// SIMATIC S7-200 project (STEP 7-Micro/WIN), CPU 226 REL 02.01

SYMBOL_TABLE 用户定义1
DDL              I0.0     // 压力继电器1
DDR              I0.1     // 压力继电器2
HP1              I0.2     // 正转水平位置
HP2              I0.3     // 反转水平位置
VP               I0.4     // 竖直位置
LMT1             I0.5     // 极限位置1
LMT2             I0.6     // 极限位置2
ERR              I0.7     // 急停或故障
TR               I1.2     // 正转点动
RT               I1.3     // 反转点动
HR1              I1.4     // 正转到水平
HR2              I1.5     // 反转到水平
TMP              M0.0     // 临时变量
FlagTR           M0.1     // 正转点动指令
FlagRT           M0.2     // 反转点动指令
FlagTRC          M0.3     // 正转到水平位置指令
FlagRTC          M0.4     // 反转到水平位置指令
EV1              Q0.0     // EV1
EV2              Q0.1     // EV2
EV3              Q0.2     // EV3
EV4              Q0.3     // EV4
EV5              Q0.4     // EV5
EV6              Q0.5     // EV6
EV7              Q0.6     // EV7
EV8              Q0.7     // EV8
AL1              Q1.0     // 翻转运行指示
AL2              Q1.1     // 系统运行指示
END_SYMBOL_TABLE

SYMBOL_TABLE S7-200 符号
Always_On        SM0.0    // 始终接通为 ON
First_Scan_On    SM0.1    // 仅第一个扫描周期中接通为 ON
END_SYMBOL_TABLE

ORGANIZATION_BLOCK 主程序:OB1
TITLE=程序注释
VAR
Flag_HR1_Enabled:BOOL;	// L0.0 一键转到水平位置1触发
Flag_HR2_Enabled:BOOL;	// L0.1 一键转到水平位置2触发
State_CurPosition:BYTE;	// LB1 当前位置
Cmd_TRC:BOOL;	// L2.0 
Cmd_RTC:BOOL;	// L2.1 
END_VAR
BEGIN
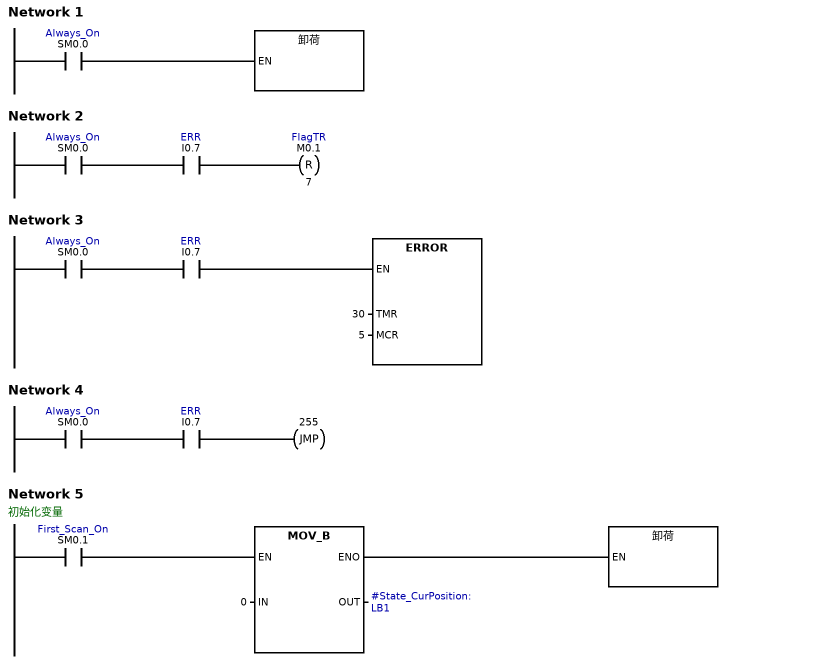
Network 1
LD     Always_On:SM0.0
CALL   卸荷:SBR0
Network 2
LD     Always_On:SM0.0
A      ERR:I0.7
R      FlagTR:M0.1, 7
Network 3
LD     Always_On:SM0.0
A      ERR:I0.7
CALL   ERROR:SBR8, 30, 5
Network 4
LD     Always_On:SM0.0
A      ERR:I0.7
JMP    255
Network 5
// 初始化变量
LD     First_Scan_On:SM0.1
MOVB   0, #State_CurPosition:LB1
AENO
CALL   卸荷:SBR0
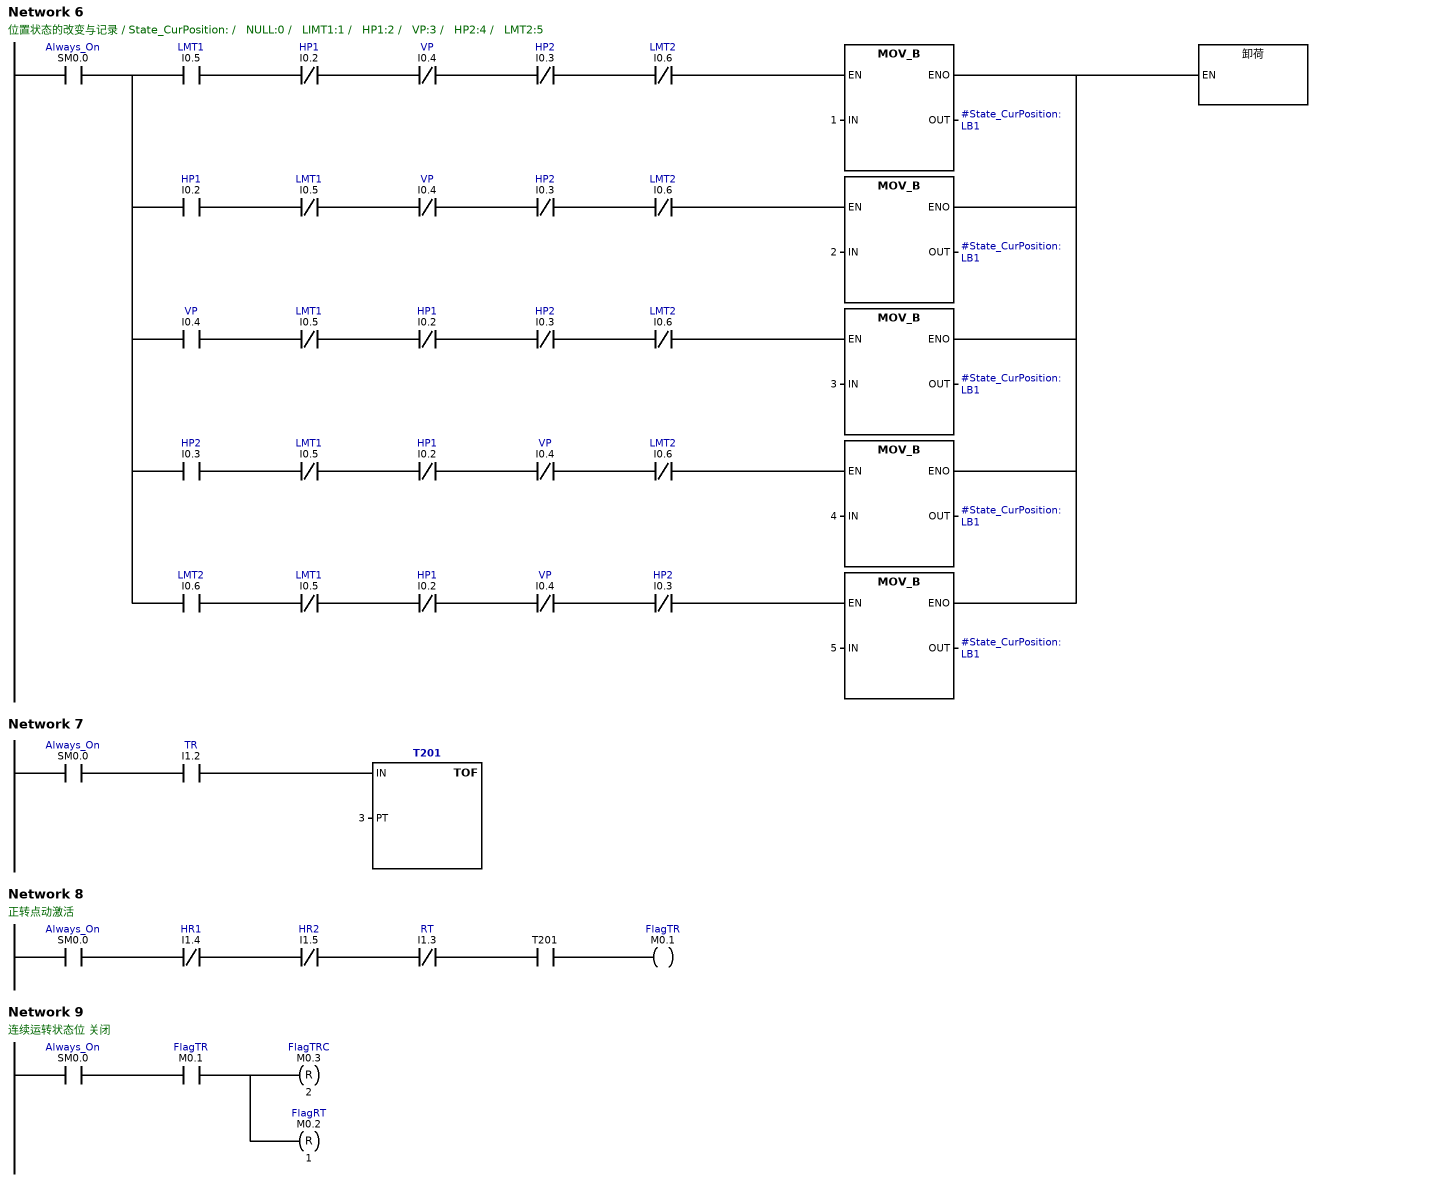
Network 6
// 位置状态的改变与记录
// State_CurPosition:
// 	NULL:0
// 	LIMT1:1
// 	HP1:2
// 	VP:3
// 	HP2:4
// 	LMT2:5
LD     Always_On:SM0.0
LPS
A      LMT1:I0.5
AN     HP1:I0.2
AN     VP:I0.4
AN     HP2:I0.3
AN     LMT2:I0.6
MOVB   1, #State_CurPosition:LB1
AENO
=      L63.7
LRD
A      HP1:I0.2
AN     LMT1:I0.5
AN     VP:I0.4
AN     HP2:I0.3
AN     LMT2:I0.6
MOVB   2, #State_CurPosition:LB1
AENO
O      L63.7
=      L63.6
LRD
A      VP:I0.4
AN     LMT1:I0.5
AN     HP1:I0.2
AN     HP2:I0.3
AN     LMT2:I0.6
MOVB   3, #State_CurPosition:LB1
AENO
O      L63.6
=      L63.5
LRD
A      HP2:I0.3
AN     LMT1:I0.5
AN     HP1:I0.2
AN     VP:I0.4
AN     LMT2:I0.6
MOVB   4, #State_CurPosition:LB1
AENO
O      L63.5
=      L63.4
LPP
A      LMT2:I0.6
AN     LMT1:I0.5
AN     HP1:I0.2
AN     VP:I0.4
AN     HP2:I0.3
MOVB   5, #State_CurPosition:LB1
AENO
O      L63.4
CALL   卸荷:SBR0
Network 7
LD     Always_On:SM0.0
A      TR:I1.2
TOF    T201, 3
Network 8
// 正转点动激活
LD     Always_On:SM0.0
AN     HR1:I1.4
AN     HR2:I1.5
AN     RT:I1.3
A      T201
=      FlagTR:M0.1
Network 9
// 连续运转状态位 关闭
LD     Always_On:SM0.0
A      FlagTR:M0.1
R      FlagTRC:M0.3, 2
R      FlagRT:M0.2, 1
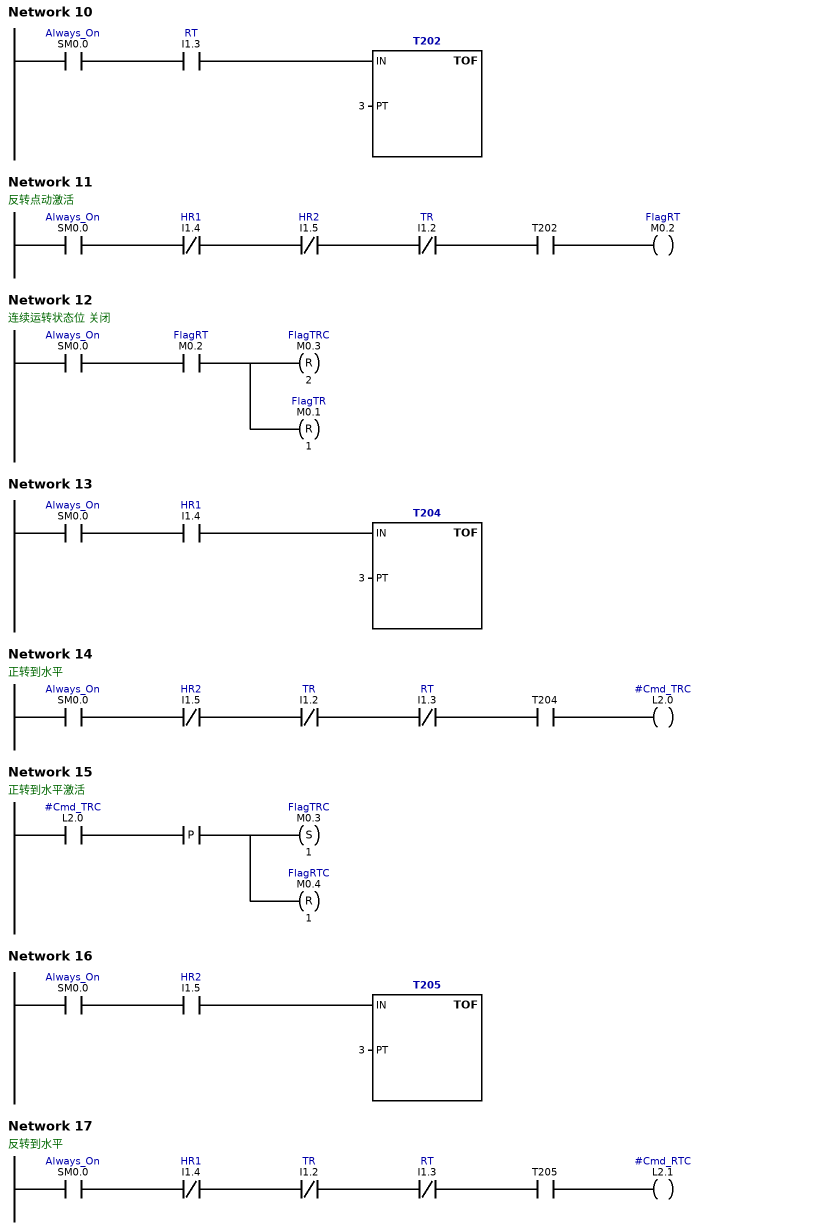
Network 10
LD     Always_On:SM0.0
A      RT:I1.3
TOF    T202, 3
Network 11
// 反转点动激活
LD     Always_On:SM0.0
AN     HR1:I1.4
AN     HR2:I1.5
AN     TR:I1.2
A      T202
=      FlagRT:M0.2
Network 12
// 连续运转状态位 关闭
LD     Always_On:SM0.0
A      FlagRT:M0.2
R      FlagTRC:M0.3, 2
R      FlagTR:M0.1, 1
Network 13
LD     Always_On:SM0.0
A      HR1:I1.4
TOF    T204, 3
Network 14
// 正转到水平
LD     Always_On:SM0.0
AN     HR2:I1.5
AN     TR:I1.2
AN     RT:I1.3
A      T204
=      #Cmd_TRC:L2.0
Network 15
// 正转到水平激活
LD     #Cmd_TRC:L2.0
EU
S      FlagTRC:M0.3, 1
R      FlagRTC:M0.4, 1
Network 16
LD     Always_On:SM0.0
A      HR2:I1.5
TOF    T205, 3
Network 17
// 反转到水平
LD     Always_On:SM0.0
AN     HR1:I1.4
AN     TR:I1.2
AN     RT:I1.3
A      T205
=      #Cmd_RTC:L2.1
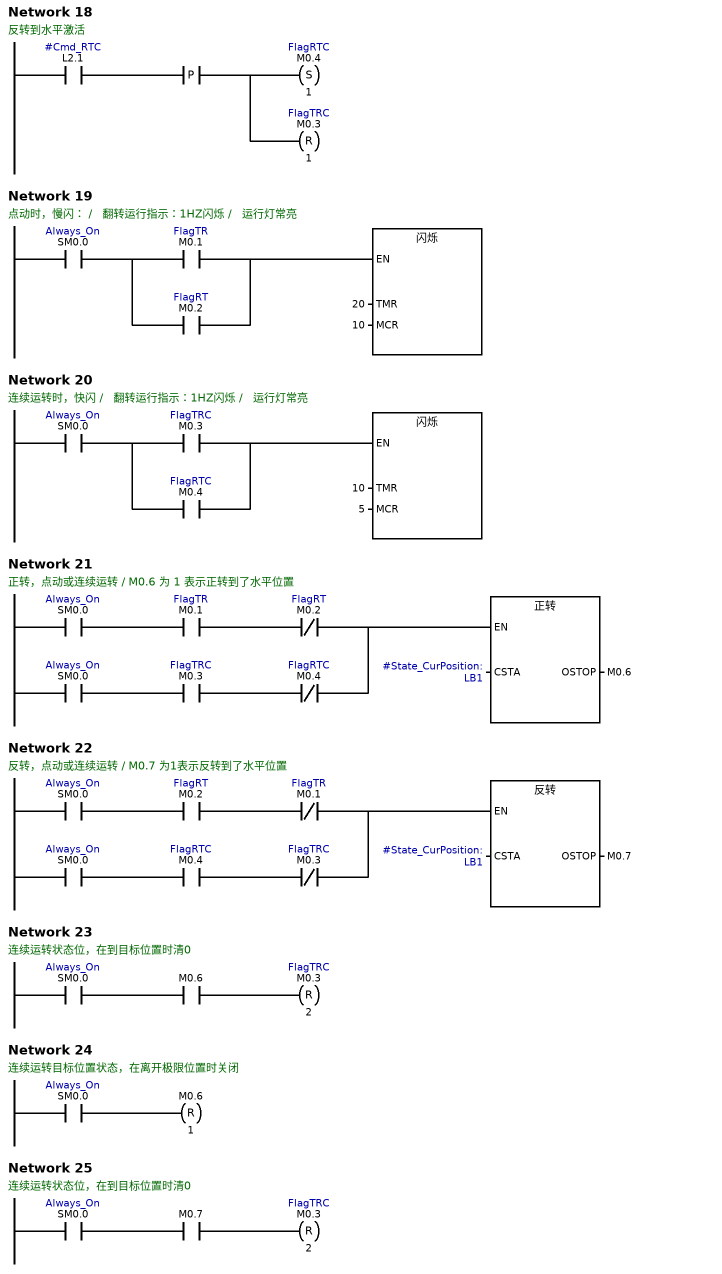
Network 18
// 反转到水平激活
LD     #Cmd_RTC:L2.1
EU
S      FlagRTC:M0.4, 1
R      FlagTRC:M0.3, 1
Network 19
// 点动时，慢闪：
// 	翻转运行指示：1HZ闪烁
// 	运行灯常亮
LD     Always_On:SM0.0
LD     FlagTR:M0.1
O      FlagRT:M0.2
ALD
CALL   闪烁:SBR3, 20, 10
Network 20
// 连续运转时，快闪
// 	翻转运行指示：1HZ闪烁
// 	运行灯常亮
LD     Always_On:SM0.0
LD     FlagTRC:M0.3
O      FlagRTC:M0.4
ALD
CALL   闪烁:SBR3, 10, 5
Network 21
// 正转，点动或连续运转
// M0.6 为 1 表示正转到了水平位置
LD     Always_On:SM0.0
A      FlagTR:M0.1
AN     FlagRT:M0.2
LD     Always_On:SM0.0
A      FlagTRC:M0.3
AN     FlagRTC:M0.4
OLD
CALL   正转:SBR1, #State_CurPosition:LB1, M0.6
Network 22
// 反转，点动或连续运转
// M0.7 为1表示反转到了水平位置
LD     Always_On:SM0.0
A      FlagRT:M0.2
AN     FlagTR:M0.1
LD     Always_On:SM0.0
A      FlagRTC:M0.4
AN     FlagTRC:M0.3
OLD
CALL   反转:SBR2, #State_CurPosition:LB1, M0.7
Network 23
// 连续运转状态位，在到目标位置时清0
LD     Always_On:SM0.0
A      M0.6
R      FlagTRC:M0.3, 2
Network 24
// 连续运转目标位置状态，在离开极限位置时关闭
LD     Always_On:SM0.0
R      M0.6, 1
Network 25
// 连续运转状态位，在到目标位置时清0
LD     Always_On:SM0.0
A      M0.7
R      FlagTRC:M0.3, 2
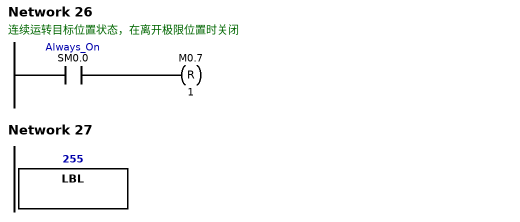
Network 26
// 连续运转目标位置状态，在离开极限位置时关闭
LD     Always_On:SM0.0
R      M0.7, 1
Network 27
LBL    255
END_ORGANIZATION_BLOCK

SUBROUTINE_BLOCK 卸荷:SBR0
TITLE=子程序注释
BEGIN
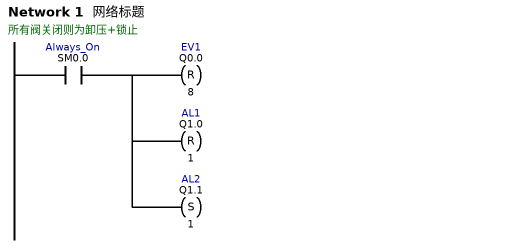
Network 1 // 网络标题
// 所有阀关闭则为卸压+锁止
LD     Always_On:SM0.0
R      EV1:Q0.0, 8
R      AL1:Q1.0, 1
S      AL2:Q1.1, 1
END_SUBROUTINE_BLOCK

SUBROUTINE_BLOCK 正转:SBR1
TITLE=子程序注释
VAR_INPUT
CSTA:BYTE;	// LB0 
END_VAR
VAR_OUTPUT
OSTOP:BOOL;	// L1.0 
END_VAR
BEGIN
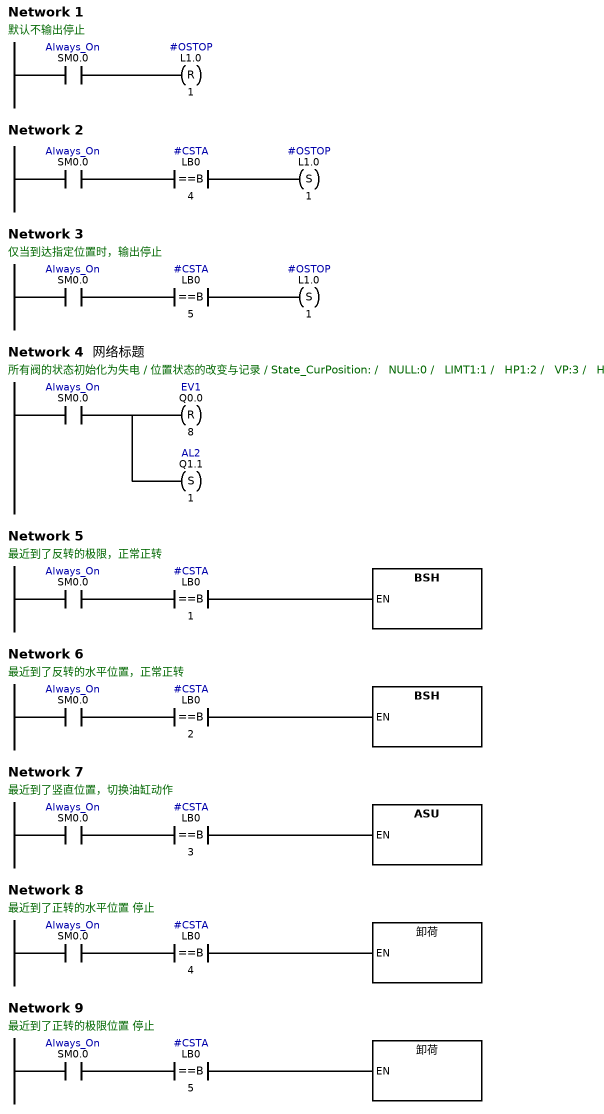
Network 1
// 默认不输出停止 
LD     Always_On:SM0.0
R      #OSTOP:L1.0, 1
Network 2
LD     Always_On:SM0.0
AB=    #CSTA:LB0, 4
S      #OSTOP:L1.0, 1
Network 3
// 仅当到达指定位置时，输出停止
LD     Always_On:SM0.0
AB=    #CSTA:LB0, 5
S      #OSTOP:L1.0, 1
Network 4 // 网络标题
// 所有阀的状态初始化为失电
// 位置状态的改变与记录
// State_CurPosition:
// 	NULL:0
// 	LIMT1:1
// 	HP1:2
// 	VP:3
// 	HP2:4
// 	LMT2:5
LD     Always_On:SM0.0
R      EV1:Q0.0, 8
S      AL2:Q1.1, 1
Network 5
// 最近到了反转的极限，正常正转
LD     Always_On:SM0.0
AB=    #CSTA:LB0, 1
CALL   BSH:SBR5
Network 6
// 最近到了反转的水平位置，正常正转
LD     Always_On:SM0.0
AB=    #CSTA:LB0, 2
CALL   BSH:SBR5
Network 7
// 最近到了竖直位置，切换油缸动作
LD     Always_On:SM0.0
AB=    #CSTA:LB0, 3
CALL   ASU:SBR6
Network 8
// 最近到了正转的水平位置 停止
LD     Always_On:SM0.0
AB=    #CSTA:LB0, 4
CALL   卸荷:SBR0
Network 9
// 最近到了正转的极限位置 停止
LD     Always_On:SM0.0
AB=    #CSTA:LB0, 5
CALL   卸荷:SBR0
END_SUBROUTINE_BLOCK

SUBROUTINE_BLOCK 反转:SBR2
TITLE=
VAR_INPUT
CSTA:BYTE;	// LB0 
END_VAR
VAR_OUTPUT
OSTOP:BOOL;	// L1.0 
END_VAR
BEGIN
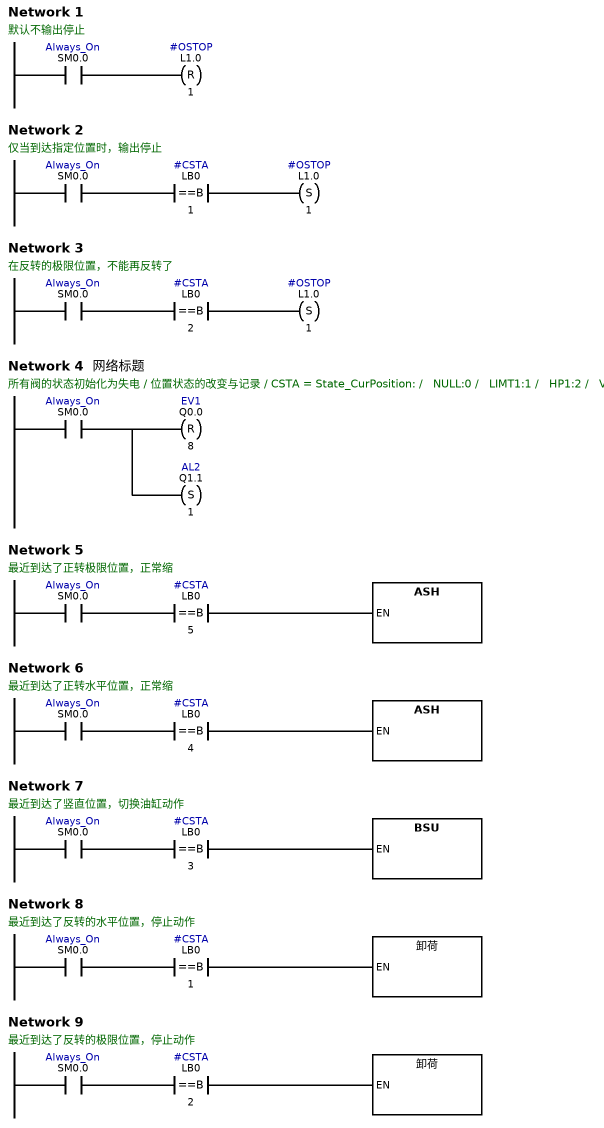
Network 1
// 默认不输出停止 
LD     Always_On:SM0.0
R      #OSTOP:L1.0, 1
Network 2
// 仅当到达指定位置时，输出停止
LD     Always_On:SM0.0
AB=    #CSTA:LB0, 1
S      #OSTOP:L1.0, 1
Network 3
// 在反转的极限位置，不能再反转了
LD     Always_On:SM0.0
AB=    #CSTA:LB0, 2
S      #OSTOP:L1.0, 1
Network 4 // 网络标题
// 所有阀的状态初始化为失电
// 位置状态的改变与记录
// CSTA = State_CurPosition:
// 	NULL:0
// 	LIMT1:1
// 	HP1:2
// 	VP:3
// 	HP2:4
// 	LMT2:5
LD     Always_On:SM0.0
R      EV1:Q0.0, 8
S      AL2:Q1.1, 1
Network 5
// 最近到达了正转极限位置，正常缩
LD     Always_On:SM0.0
AB=    #CSTA:LB0, 5
CALL   ASH:SBR4
Network 6
// 最近到达了正转水平位置，正常缩
LD     Always_On:SM0.0
AB=    #CSTA:LB0, 4
CALL   ASH:SBR4
Network 7
// 最近到达了竖直位置，切换油缸动作
LD     Always_On:SM0.0
AB=    #CSTA:LB0, 3
CALL   BSU:SBR7
Network 8
// 最近到达了反转的水平位置，停止动作
LD     Always_On:SM0.0
AB=    #CSTA:LB0, 1
CALL   卸荷:SBR0
Network 9
// 最近到达了反转的极限位置，停止动作
LD     Always_On:SM0.0
AB=    #CSTA:LB0, 2
CALL   卸荷:SBR0
END_SUBROUTINE_BLOCK

SUBROUTINE_BLOCK 闪烁:SBR3
TITLE=
VAR_INPUT
TMR:INT;	// LW0 
MCR:INT;	// LW2 
END_VAR
BEGIN
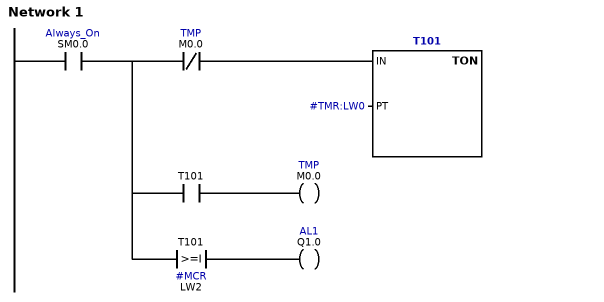
Network 1
LD     Always_On:SM0.0
LPS
AN     TMP:M0.0
TON    T101, #TMR:LW0
LRD
A      T101
=      TMP:M0.0
LPP
AW>=   T101, #MCR:LW2
=      AL1:Q1.0
END_SUBROUTINE_BLOCK

SUBROUTINE_BLOCK ASH:SBR4
TITLE=子程序注释
VAR
RUN:BOOL;	// L0.0 
END_VAR
BEGIN
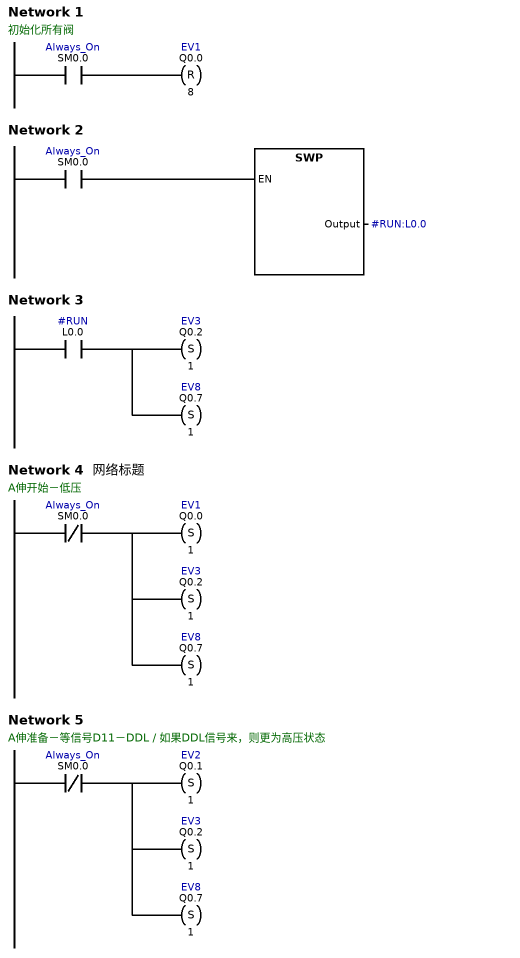
Network 1
// 初始化所有阀
LD     Always_On:SM0.0
R      EV1:Q0.0, 8
Network 2
LD     Always_On:SM0.0
CALL   SWP:SBR9, #RUN:L0.0
Network 3
LD     #RUN:L0.0
S      EV3:Q0.2, 1
S      EV8:Q0.7, 1
Network 4 // 网络标题
// A伸开始－低压
LDN    Always_On:SM0.0
S      EV1:Q0.0, 1
S      EV3:Q0.2, 1
S      EV8:Q0.7, 1
Network 5
// A伸准备－等信号D11－DDL
// 如果DDL信号来，则更为高压状态
LDN    Always_On:SM0.0
S      EV2:Q0.1, 1
S      EV3:Q0.2, 1
S      EV8:Q0.7, 1
END_SUBROUTINE_BLOCK

SUBROUTINE_BLOCK BSH:SBR5
TITLE=
VAR
RUN:BOOL;	// L0.0 
END_VAR
BEGIN
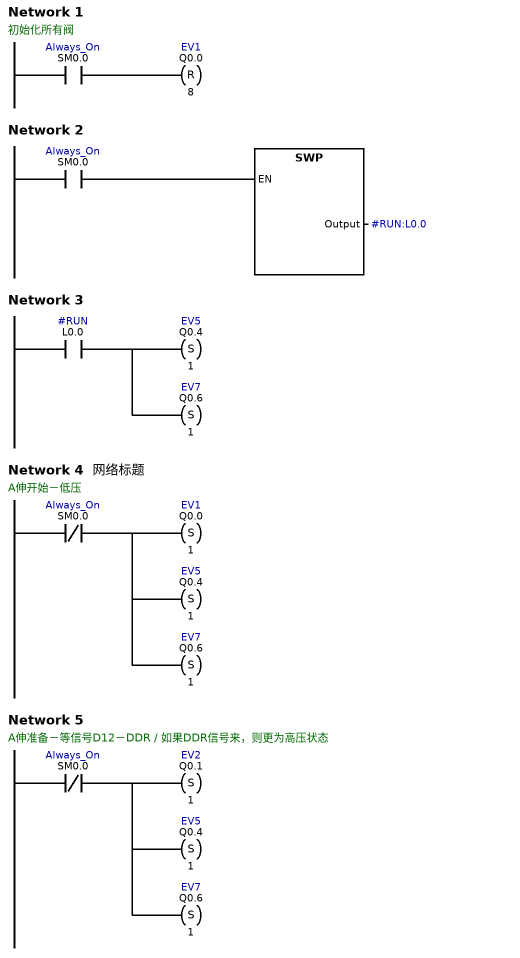
Network 1
// 初始化所有阀
LD     Always_On:SM0.0
R      EV1:Q0.0, 8
Network 2
LD     Always_On:SM0.0
CALL   SWP:SBR9, #RUN:L0.0
Network 3
LD     #RUN:L0.0
S      EV5:Q0.4, 1
S      EV7:Q0.6, 1
Network 4 // 网络标题
// A伸开始－低压
LDN    Always_On:SM0.0
S      EV1:Q0.0, 1
S      EV5:Q0.4, 1
S      EV7:Q0.6, 1
Network 5
// A伸准备－等信号D12－DDR
// 如果DDR信号来，则更为高压状态
LDN    Always_On:SM0.0
S      EV2:Q0.1, 1
S      EV5:Q0.4, 1
S      EV7:Q0.6, 1
END_SUBROUTINE_BLOCK

SUBROUTINE_BLOCK ASU:SBR6
TITLE=
VAR
RUN:BOOL;	// L0.0 
END_VAR
BEGIN
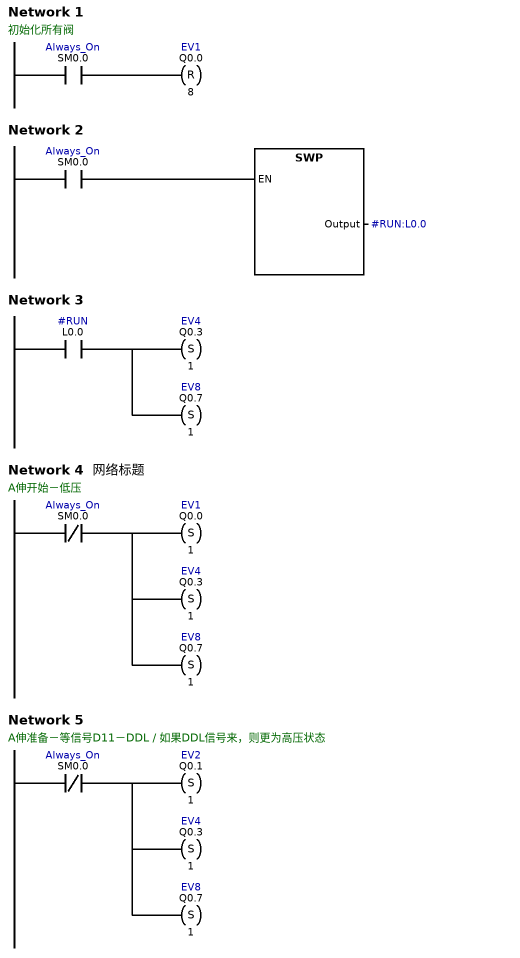
Network 1
// 初始化所有阀
LD     Always_On:SM0.0
R      EV1:Q0.0, 8
Network 2
LD     Always_On:SM0.0
CALL   SWP:SBR9, #RUN:L0.0
Network 3
LD     #RUN:L0.0
S      EV4:Q0.3, 1
S      EV8:Q0.7, 1
Network 4 // 网络标题
// A伸开始－低压
LDN    Always_On:SM0.0
S      EV1:Q0.0, 1
S      EV4:Q0.3, 1
S      EV8:Q0.7, 1
Network 5
// A伸准备－等信号D11－DDL
// 如果DDL信号来，则更为高压状态
LDN    Always_On:SM0.0
S      EV2:Q0.1, 1
S      EV4:Q0.3, 1
S      EV8:Q0.7, 1
END_SUBROUTINE_BLOCK

SUBROUTINE_BLOCK BSU:SBR7
TITLE=
VAR
RUN:BOOL;	// L0.0 
END_VAR
BEGIN
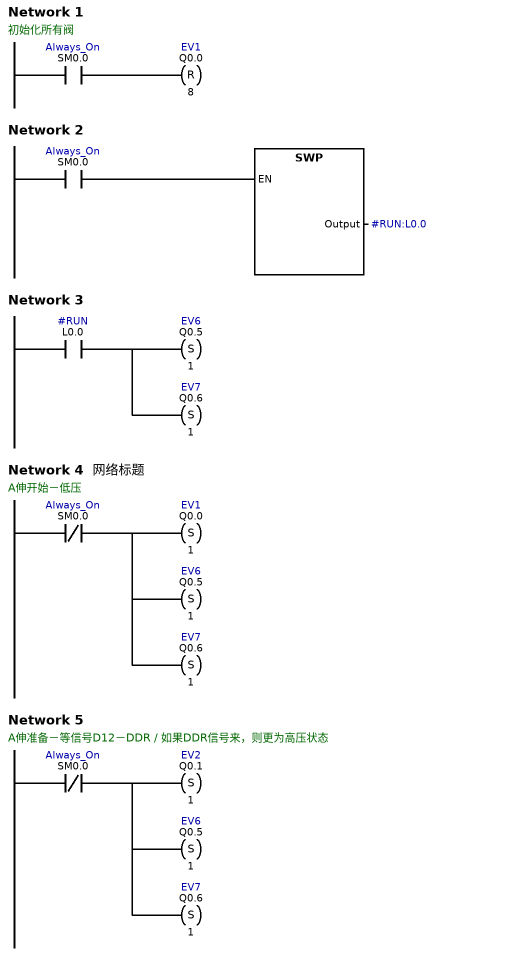
Network 1
// 初始化所有阀
LD     Always_On:SM0.0
R      EV1:Q0.0, 8
Network 2
LD     Always_On:SM0.0
CALL   SWP:SBR9, #RUN:L0.0
Network 3
LD     #RUN:L0.0
S      EV6:Q0.5, 1
S      EV7:Q0.6, 1
Network 4 // 网络标题
// A伸开始－低压
LDN    Always_On:SM0.0
S      EV1:Q0.0, 1
S      EV6:Q0.5, 1
S      EV7:Q0.6, 1
Network 5
// A伸准备－等信号D12－DDR
// 如果DDR信号来，则更为高压状态
LDN    Always_On:SM0.0
S      EV2:Q0.1, 1
S      EV6:Q0.5, 1
S      EV7:Q0.6, 1
END_SUBROUTINE_BLOCK

SUBROUTINE_BLOCK ERROR:SBR8
TITLE=子程序注释
VAR_INPUT
TMR:INT;	// LW0 
MCR:INT;	// LW2 
END_VAR
BEGIN
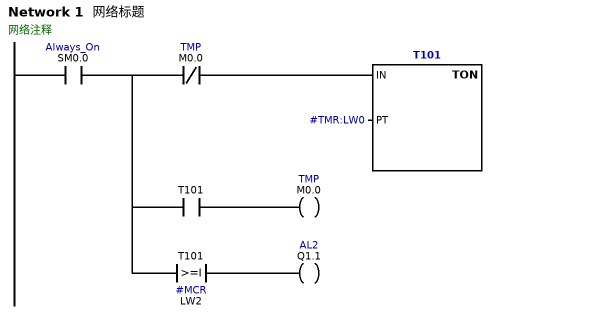
Network 1 // 网络标题
// 网络注释
LD     Always_On:SM0.0
LPS
AN     TMP:M0.0
TON    T101, #TMR:LW0
LRD
A      T101
=      TMP:M0.0
LPP
AW>=   T101, #MCR:LW2
=      AL2:Q1.1
END_SUBROUTINE_BLOCK

SUBROUTINE_BLOCK SWP:SBR9
TITLE=子程序注释
VAR_OUTPUT
Output:BOOL;	// L0.0 
END_VAR
BEGIN
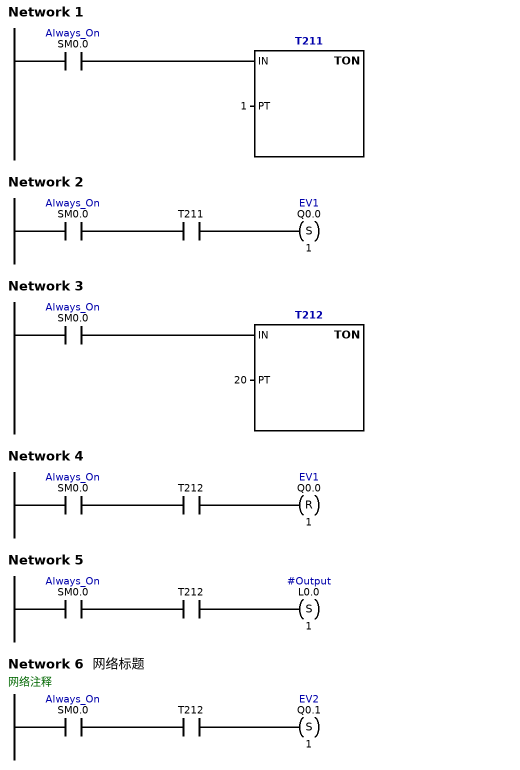
Network 1
LD     Always_On:SM0.0
TON    T211, 1
Network 2
LD     Always_On:SM0.0
A      T211
S      EV1:Q0.0, 1
Network 3
LD     Always_On:SM0.0
TON    T212, 20
Network 4
LD     Always_On:SM0.0
A      T212
R      EV1:Q0.0, 1
Network 5
LD     Always_On:SM0.0
A      T212
S      #Output:L0.0, 1
Network 6 // 网络标题
// 网络注释
LD     Always_On:SM0.0
A      T212
S      EV2:Q0.1, 1
END_SUBROUTINE_BLOCK

DATA_BLOCK_TAB 用户定义1
BEGIN
//数据页注释
//按 F1 键获取帮助和示范数据页
VB0      255
VB1      255
VB2      255
END_DATA_BLOCK_TAB
